SUBAPPLICATION IXA_TO_Aux_QXA (* logiBUS_IXA auf isobus Aux_QXA (generisch), adapter-basiert *)
  (* Standard: 61499-2 *)
  (* Version 1.1, 2026-09-18, Franz Höpfinger, Meisterschulen am Ostbahnhof, IX.INITO auf IX.REQ zurueckverdrahtet (Selfloop) - loest nach der Initialisierung sofort einen Service-Request aus, statt auf die erste echte Wertaenderung am Bus zu warten (Fix fuer 'Waiting for handle'-Status direkt nach Boot). *)
  (* Version 1.0, 2026-09-09, Franz Höpfinger, Meisterschulen am Ostbahnhof, Ausgelagert aus Uebung_003c_sub_AX zur Wiederverwendung. *)
  PACKAGE MyLib::sys;
  IMPORT logiBUS::io::DI::logiBUS_DI::Invalid;
  IMPORT logiBUS::io::DI::logiBUS_DI_S;
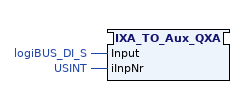
  VAR_INPUT
    Input : logiBUS::io::DI::logiBUS_DI_S := Invalid; (* Identify the Input Input_I1..I8 *)
    iInpNr : USINT := 0; (* Number of auxiliary array - corresponds with the order in the pool that means first aux input in pool is iInpNr = 0 etc. *)
  END_VAR
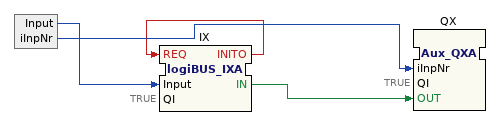
  FBS
    QX : isobus::UT::io::Auxiliary::OUT::Aux_QXA(QI := TRUE);
    IX : logiBUS::io::DI::logiBUS_IXA(QI := TRUE);
  END_FBS
  EVENT_CONNECTIONS
    IX.INITO TO IX.REQ;
  END_CONNECTIONS
  DATA_CONNECTIONS
    Input TO IX.Input;
    iInpNr TO QX.iInpNr;
  END_CONNECTIONS
  ADAPTER_CONNECTIONS
    IX.IN TO QX.OUT;
  END_CONNECTIONS
END_SUBAPPLICATION
